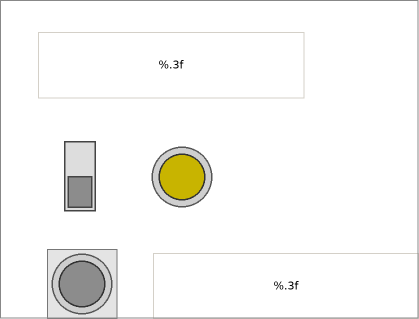
VISUALIZATION moveAbs  // 419x319
    Textfield (38,32 266x66), "%.3f", text variable: motionChalleng_moveAbs.myAxis.NcToPlc.ActPos
    DipSwitch (45,141 70x70), variable: motionChalleng_moveAbs.enableAxis, behaviour: TOGGLE, style: Switch-DipSwitch-Gray
    Lamp1 (147,142 70x70), variable: motionChalleng_moveAbs.mcPower.Status, style: Lamp-Lamp1-Yellow
    PushSwitch (47,249 70x70), variable: motionChalleng_moveAbs.executeMoveAbs, behaviour: TOGGLE, style: Switch-PushSwitch-Gray
    Textfield (153,253 266x66), "%.3f", text variable: motionChalleng_moveAbs.userSetPoint
        OnMouseDown: write motionChalleng_moveAbs.userSetPoint via Default
END_VISUALIZATION

(* stored: Version 1.1.0.1, ProductVersion 3.1.4024.5
   Visu moveAbs: Id {043ad3ad-6a15-48c5-9794-9e4865ca469c} *)
